FUNCTION_BLOCK CNVG_MDLL (* Locally-Coupled Conveyor Model with Gate for 1 Workpiece *)
  (* Standard: 61499-1; Classification: Model; ApplicationDomain: Simulation; Function: Material Handling; Type: Conveyor *)
  (* Version 0.0, 2004-10-28, JHC, Rockwell Automation, Renamed from old CNV_MDLL. *)
  (* Compiler header: package fb.rt.mva; import fb.rt.math.*; import fb.rt.net.*; *)
  (* Compiler classdef: public class CNVG_MDLL extends FBMVCD *)
  (* Compiler Java Sun JDK 1.4.2 *)
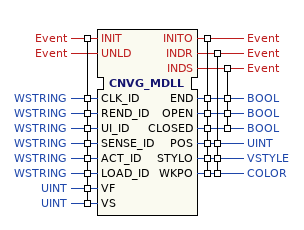
  EVENT_INPUT
    INIT WITH REND_ID, ACT_ID, VF, CLK_ID, UI_ID, SENSE_ID, VS, LOAD_ID; (* Initialize *)
    UNLD; (* Unload Workpiece if at END position *)
  END_EVENT
  EVENT_OUTPUT
    INITO WITH POS, STYLO, WKPO, END, OPEN, CLOSED; (* View Initialized *)
    INDR WITH POS, STYLO, WKPO; (* Change in Rendering Data *)
    INDS WITH END, OPEN, CLOSED; (* Change in Sensor Data *)
  END_EVENT
  VAR_INPUT
    CLK_ID : WSTRING := "SIM_CLK"; (* Simulation clock channel ID *)
    REND_ID : WSTRING; (* Rendering data channel ID to View *)
    UI_ID : WSTRING; (* User input channel ID from View *)
    SENSE_ID : WSTRING; (* Sensor data channel ID to Controller *)
    ACT_ID : WSTRING; (* Actuator data channel ID from Controller *)
    LOAD_ID : WSTRING; (* Loader channel ID for LPOS,STYLE, WKPC *)
    VF : UINT := 5; (* Conveyor Speed in % per CLK event *)
    VS : UINT := 50; (* Stopper Speed in % per CLK event *)
  END_VAR
  VAR_OUTPUT
    END : BOOL; (* Workpiece at End Position *)
    OPEN : BOOL; (* Stopper/Gate Open *)
    CLOSED : BOOL; (* Stopper/Gate Closed *)
    POS : UINT; (* Workpiece position, 0-100% *)
    STYLO : VSTYLE; (* Currently loaded workpiece style *)
    WKPO : COLOR; (* Currently loaded workpiece color *)
  END_VAR
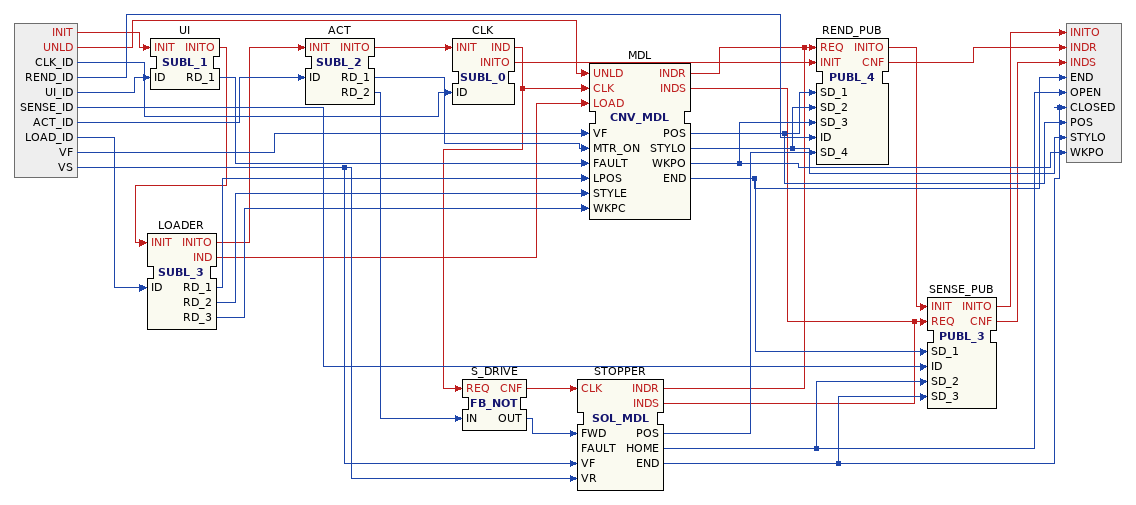
  FBS
    ACT : SUBL_2;
    MDL : CNV_MDL;
    REND_PUB : PUBL_4;
    CLK : SUBL_0;
    UI : SUBL_1;
    SENSE_PUB : PUBL_3;
    STOPPER : SOL_MDL;
    S_DRIVE : FB_NOT; (* Normal Stopper/Gate Position = CLOSED *)
    LOADER : SUBL_3;
  END_FBS
  EVENT_CONNECTIONS
    UNLD TO MDL.UNLD;
    MDL.INDR TO REND_PUB.REQ;
    CLK.IND TO MDL.CLK;
    INIT TO UI.INIT;
    ACT.INITO TO CLK.INIT;
    CLK.INITO TO REND_PUB.INIT;
    REND_PUB.INITO TO SENSE_PUB.INIT;
    SENSE_PUB.INITO TO INITO;
    SENSE_PUB.CNF TO INDS;
    MDL.INDS TO SENSE_PUB.REQ;
    REND_PUB.CNF TO INDR;
    STOPPER.INDS TO SENSE_PUB.REQ;
    CLK.IND TO S_DRIVE.REQ;
    S_DRIVE.CNF TO STOPPER.CLK;
    STOPPER.INDR TO REND_PUB.REQ;
    UI.INITO TO LOADER.INIT;
    LOADER.INITO TO ACT.INIT;
    LOADER.IND TO MDL.LOAD;
  END_CONNECTIONS
  DATA_CONNECTIONS
    MDL.POS TO REND_PUB.SD_1;
    MDL.STYLO TO REND_PUB.SD_2;
    MDL.WKPO TO REND_PUB.SD_3;
    ACT_ID TO ACT.ID;
    MDL.STYLO TO STYLO;
    MDL.WKPO TO WKPO;
    REND_ID TO REND_PUB.ID;
    MDL.POS TO POS;
    VF TO MDL.VF;
    ACT.RD_1 TO MDL.MTR_ON;
    CLK_ID TO CLK.ID;
    UI_ID TO UI.ID;
    UI.RD_1 TO MDL.FAULT;
    MDL.END TO SENSE_PUB.SD_1;
    MDL.END TO END;
    SENSE_ID TO SENSE_PUB.ID;
    STOPPER.POS TO REND_PUB.SD_4;
    STOPPER.HOME TO SENSE_PUB.SD_2;
    VS TO STOPPER.VF;
    VS TO STOPPER.VR;
    STOPPER.END TO SENSE_PUB.SD_3;
    STOPPER.HOME TO OPEN;
    STOPPER.END TO CLOSED;
    S_DRIVE.OUT TO STOPPER.FWD;
    ACT.RD_2 TO S_DRIVE.IN;
    LOADER.RD_1 TO MDL.LPOS;
    LOADER.RD_2 TO MDL.STYLE;
    LOADER.RD_3 TO MDL.WKPC;
    LOAD_ID TO LOADER.ID;
  END_CONNECTIONS
END_FUNCTION_BLOCK
